TYPE OutputBase_10CEE7DE :
STRUCT
END_STRUCT
END_TYPE

(* stored: Version 1.2.0.0, ProductVersion 3.1.4024.12
   DUT OutputBase_10CEE7DE: Id {26488daa-16a9-0777-2bd0-7dcb9534b4e6} *)
